// Mitsubishi GX Developer project: ハンドル角入力部_originalPLC   PLC: FX2N

PROGRAM MAIN
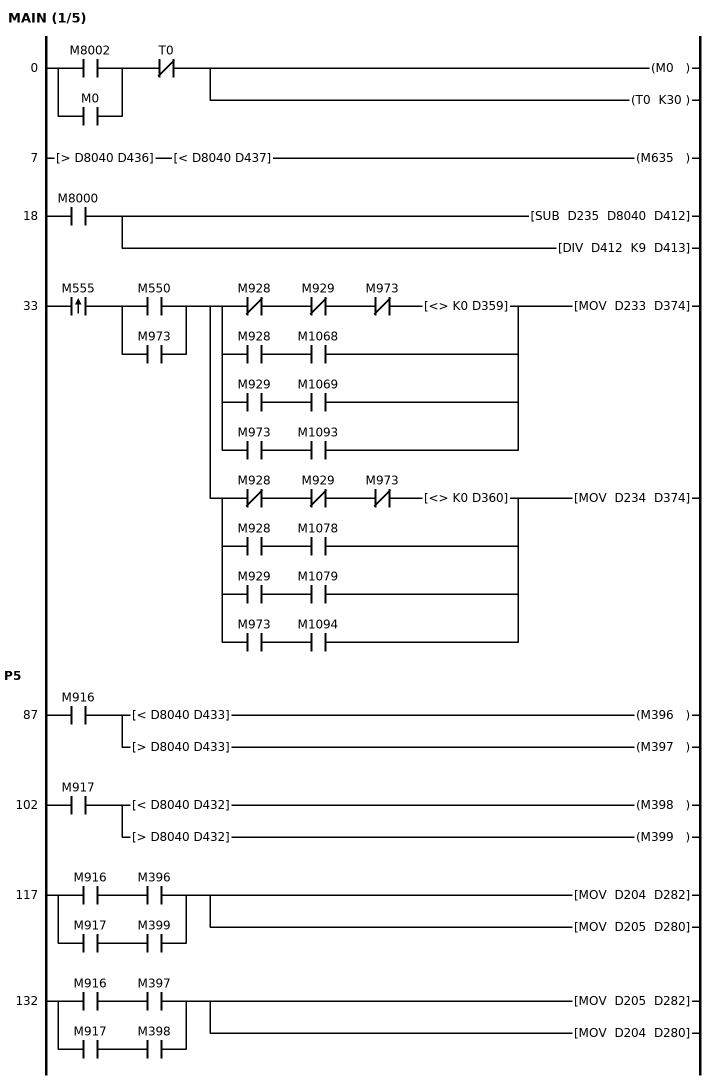
0     LD      M8002
      OR      M0
      ANI     T0
      OUT     M0
      OUT     T0 K30
7     LD>     D8040 D436
      AND<    D8040 D437
      OUT     M635
18    LD      M8000
      SUB     D235 D8040 D412
      DIV     D412 K9 D413
33    LDP     M555
      LD      M550
      OR      M973
      ANB
      MPS
      LDI     M928
      ANI     M929
      ANI     M973
      AND<>   K0 D359
      LD      M928
      AND     M1068
      ORB
      LD      M929
      AND     M1069
      ORB
      LD      M973
      AND     M1093
      ORB
      ANB
      MOV     D233 D374
      MPP
      LDI     M928
      ANI     M929
      ANI     M973
      AND<>   K0 D360
      LD      M928
      AND     M1078
      ORB
      LD      M929
      AND     M1079
      ORB
      LD      M973
      AND     M1094
      ORB
      ANB
      MOV     D234 D374
      P5
87    LD      M916
      MPS
      AND<    D8040 D433
      OUT     M396
      MPP
      AND>    D8040 D433
      OUT     M397
102   LD      M917
      MPS
      AND<    D8040 D432
      OUT     M398
      MPP
      AND>    D8040 D432
      OUT     M399
117   LD      M916
      AND     M396
      LD      M917
      AND     M399
      ORB
      MOV     D204 D282
      MOV     D205 D280
132   LD      M916
      AND     M397
      LD      M917
      AND     M398
      ORB
      MOV     D205 D282
      MOV     D204 D280
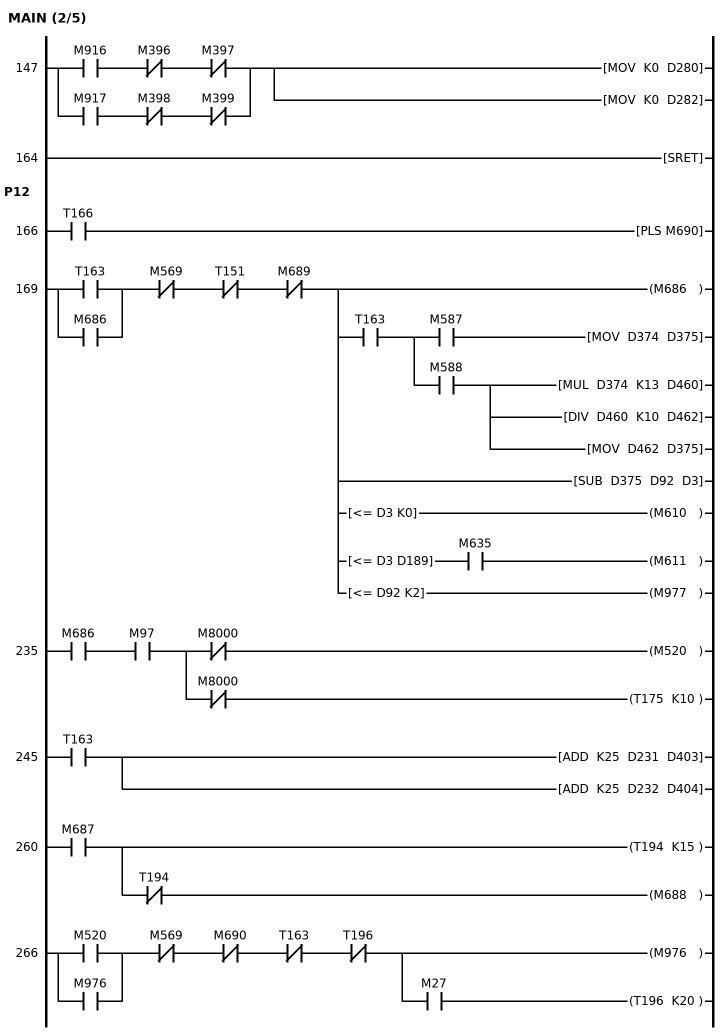
147   LD      M916
      ANI     M396
      ANI     M397
      LD      M917
      ANI     M398
      ANI     M399
      ORB
      MOV     K0 D280
      MOV     K0 D282
164   SRET
      P12
166   LD      T166
      PLS     M690
169   LD      T163
      OR      M686
      ANI     M569
      ANI     T151
      ANI     M689
      OUT     M686
      MPS
      AND     T163
      MPS
      AND     M587
      MOV     D374 D375
      MPP
      AND     M588
      MUL     D374 K13 D460
      DIV     D460 K10 D462
      MOV     D462 D375
      MPP
      SUB     D375 D92 D3
      MPS
      AND<=   D3 K0
      OUT     M610
      MRD
      AND<=   D3 D189
      AND     M635
      OUT     M611
      MPP
      AND<=   D92 K2
      OUT     M977
235   LD      M686
      AND     M97
      MPS
      ANI     M8000
      OUT     M520
      MPP
      ANI     M8000
      OUT     T175 K10
245   LD      T163
      ADD     K25 D231 D403
      ADD     K25 D232 D404
260   LD      M687
      OUT     T194 K15
      ANI     T194
      OUT     M688
266   LD      M520
      OR      M976
      ANI     M569
      ANI     M690
      ANI     T163
      ANI     T196
      OUT     M976
      AND     M27
      OUT     T196 K20
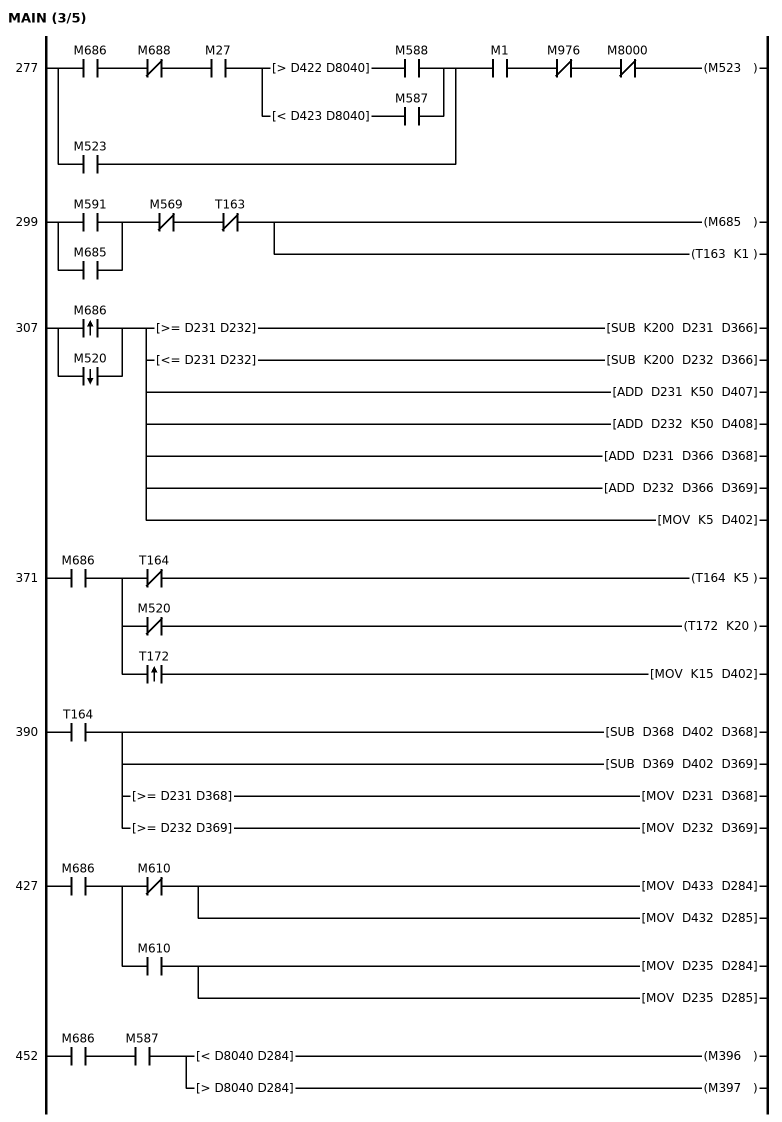
277   LD      M686
      ANI     M688
      AND     M27
      LD>     D422 D8040
      AND     M588
      LD<     D423 D8040
      AND     M587
      ORB
      ANB
      OR      M523
      AND     M1
      ANI     M976
      ANI     M8000
      OUT     M523
299   LD      M591
      OR      M685
      ANI     M569
      ANI     T163
      OUT     M685
      OUT     T163 K1
307   LDP     M686
      ORF     M520
      MPS
      AND>=   D231 D232
      SUB     K200 D231 D366
      MRD
      AND<=   D231 D232
      SUB     K200 D232 D366
      MPP
      ADD     D231 K50 D407
      ADD     D232 K50 D408
      ADD     D231 D366 D368
      ADD     D232 D366 D369
      MOV     K5 D402
371   LD      M686
      MPS
      ANI     T164
      OUT     T164 K5
      MRD
      ANI     M520
      OUT     T172 K20
      MPP
      ANDP    T172
      MOV     K15 D402
390   LD      T164
      SUB     D368 D402 D368
      SUB     D369 D402 D369
      MPS
      AND>=   D231 D368
      MOV     D231 D368
      MPP
      AND>=   D232 D369
      MOV     D232 D369
427   LD      M686
      MPS
      ANI     M610
      MOV     D433 D284
      MOV     D432 D285
      MPP
      AND     M610
      MOV     D235 D284
      MOV     D235 D285
452   LD      M686
      AND     M587
      MPS
      AND<    D8040 D284
      OUT     M396
      MPP
      AND>    D8040 D284
      OUT     M397
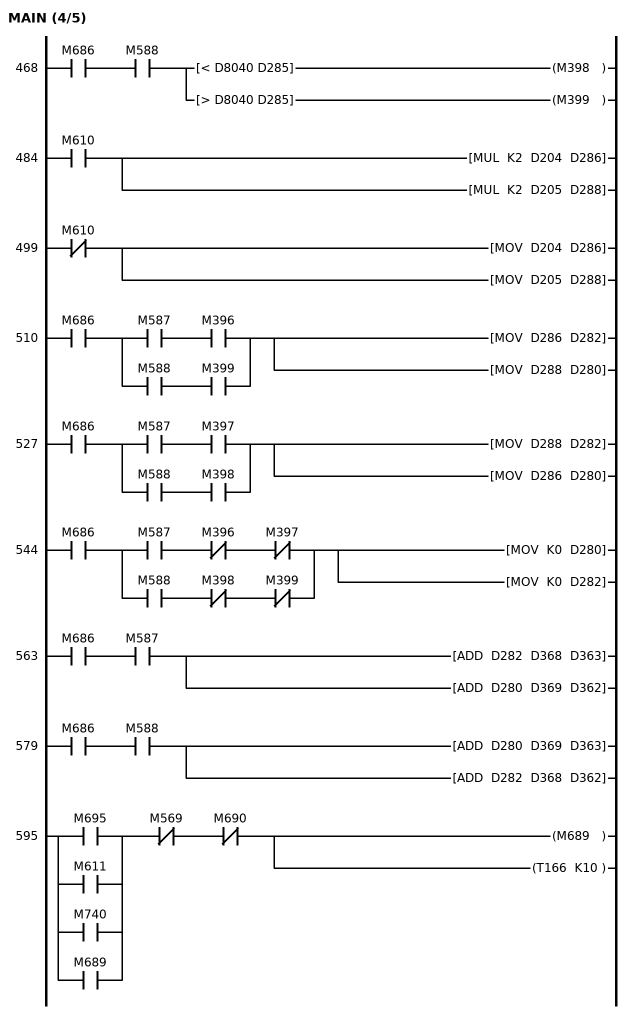
468   LD      M686
      AND     M588
      MPS
      AND<    D8040 D285
      OUT     M398
      MPP
      AND>    D8040 D285
      OUT     M399
484   LD      M610
      MUL     K2 D204 D286
      MUL     K2 D205 D288
499   LDI     M610
      MOV     D204 D286
      MOV     D205 D288
510   LD      M686
      LD      M587
      AND     M396
      LD      M588
      AND     M399
      ORB
      ANB
      MOV     D286 D282
      MOV     D288 D280
527   LD      M686
      LD      M587
      AND     M397
      LD      M588
      AND     M398
      ORB
      ANB
      MOV     D288 D282
      MOV     D286 D280
544   LD      M686
      LD      M587
      ANI     M396
      ANI     M397
      LD      M588
      ANI     M398
      ANI     M399
      ORB
      ANB
      MOV     K0 D280
      MOV     K0 D282
563   LD      M686
      AND     M587
      ADD     D282 D368 D363
      ADD     D280 D369 D362
579   LD      M686
      AND     M588
      ADD     D280 D369 D363
      ADD     D282 D368 D362
595   LD      M695
      OR      M611
      OR      M740
      OR      M689
      ANI     M569
      ANI     M690
      OUT     M689
      OUT     T166 K10
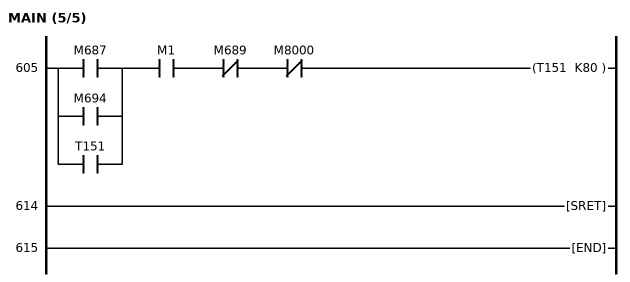
605   LD      M687
      OR      M694
      OR      T151
      AND     M1
      ANI     M689
      ANI     M8000
      OUT     T151 K80
614   SRET
615   END
END_PROGRAM
